// TIA Portal V20 export
TYPE "UDT_PartPresence"
   STRUCT
      Part : Bool;
      BW : Bool;
   END_STRUCT;
END_TYPE
